TYPE DUT_TASK :
STRUCT
	///Name of the Task
	Name: STRING[80];
	///Free to use = TRUE, busy to use =FALSE
	Dummy: BOOL := TRUE;
	///Identification number of the Task
	TaskID: INT;
	///Identification number of the Recipe
	RecipeID: INT;
	///Range of Skill in the TASK
	Skill: ARRAY[0..TaskSkillCnt] OF DUT_SKILL;
	///When occurs the action
	Timestamp: STRING[80];
	///State of the TASK e.g (unassigned, assigned, waitingForSkillReady, inProgress, done, aborted, error)
	State: DUT_TASKSTATE;
	//
	AbortTask : BOOL := FALSE;
END_STRUCT
END_TYPE

(* stored: Version 1.1.0.1, ProductVersion 3.1.0.25
   DUT DUT_TASK: Id {26ea22a7-ebc4-40c2-9ec0-99f782c1cc7a} *)
